Staubli VAL3: CutBlankLine.pgx

public program CutBlankLine(num& x_nFileId, num& x_nLine, string& x_sLine)
begin
  do
    x_nLine=$fileGet(x_nFileId,x_sLine,1)
    if x_nLine<1
      return
    endIf
    call CutSpace(x_sLine,x_sLine)
    delay(0)
  until x_sLine!=""
end
